FUNCTION_BLOCK AddRecipeToDatabase //IMPLEMENTS I_TcEventBase
VAR
	cmd : ARRAY[0..19] OF STRING_5K;
	query : STRING_5K;
	
	fbSQLCommand : FB_SQLCommandEvt(sNetID := '', tTimeout := T#5S);
	fbSQLDatabase : FB_SQLDatabaseEvt (sNetID := '', tTimeout := T#5S);
	fbSQLResult: FB_SQLResultEvt(sNetID:='', tTimeout:=T#5S);
	
	eventString : STRING_5K;
	
	step : (CONNECT, READY, EXECUTE, FINISH);
END_VAR
VAR_OUTPUT
	finished : BOOL;
END_VAR

CASE step OF
	CONNECT:
		IF fbSQLDatabase.Connect(1) THEN
			IF NOT fbSqlDatabase.bError THEN
				step := READY;
			END_IF
		END_IF
		
	READY:
		IF fbSQLDatabase.CreateCmd(ADR(fbSQLCommand)) THEN
			step := EXECUTE;
		END_IF
	
	EXECUTE:
		query := completeQuery();
		IF fbSQLCommand.Execute(ADR(query), SIZEOF(query)) THEN
			step := FINISH;
		END_IF
		
	FINISH:
		IF fbSQLDatabase.Disconnect() THEN
			finished := TRUE;
		END_IF
END_CASE

METHOD completeQuery : STRING_5K
VAR_INST
	reqProcess : ARRAY[0..3] OF STRING_5K;
	
	queryOpening : STRING_5K := 'INSERT INTO "Bundle Data - Prototype" (BundleID, Weight, Length, Height, Width, Pieces, Layers, PiecesPerLayer, ExtrusionWeight, ExtrusionHeight, ExtrusionWidth, RequiredProcesses, Paper_top, Paper_sides, Paper_bottom, Cardboard, CornerGuard, Chipboard, WoodBunk) VALUES (';;
	queryClosing : STRING_5K := ')';
END_VAR
reqProcess[0] := TO_STRING(BundleData.requiredProcessing[0]);
reqProcess[1] := TO_STRING(BundleData.requiredProcessing[1]);
reqProcess[2] := TO_STRING(BundleData.requiredProcessing[2]);
reqProcess[3] := TO_STRING(BundleData.requiredProcessing[3]);


cmd[0] := TO_STRING(BundleData.id);
CONCAT2(ADR('$''), ADR(cmd[0]), ADR(cmd[0]), SIZEOF(cmd[0]));
CONCAT2(ADR(cmd[0]), ADR('$''), ADR(cmd[0]), SIZEOF(cmd[0]));

cmd[1] := TO_STRING(BundleData.weight);
cmd[2] := TO_STRING(BundleData.length);
cmd[3] := TO_STRING(BundleData.height);
cmd[4] := TO_STRING(BundleData.width);
cmd[5] := TO_STRING(BundleData.pieces);
cmd[6] := TO_STRING(BundleData.layers);
cmd[7] := TO_STRING(BundleData.piecesPerLayer);

cmd[8] := TO_STRING(ExtrusionData.extrusionWeight);
cmd[9] := TO_STRING(ExtrusionData.extrusionHeight);
cmd[10] := TO_STRING(ExtrusionData.extrusionWidth);

cmd[11] := ConcatStrings(reqProcess, 'ARRAY[', ']', ',');
//strap wrap recipe
cmd[12] := paperQuery(StrapWrapRecipe.TopPaper); //Paper_top
cmd[13] := paperQuery(StrapWrapRecipe.LeftPaper); //Paper_sides
cmd[14] := paperQuery(StrapWrapRecipe.RightPaper); //Paper_sides
cmd[15] := paperQuery(StrapWrapRecipe.BottomPaper); //Paper_sides

cmd[16] := materialQuery(StrapWrapRecipe.Cardboard);
cmd[17] := materialQuery(StrapWrapRecipe.CornerGuard);
cmd[18] := materialQuery(StrapWrapRecipe.Chipboard);
cmd[19] := materialQuery(StrapWrapRecipe.WoodBunk);

completeQuery := ConcatStrings(cmd, queryOpening, queryClosing, ',');
END_METHOD

METHOD materialQuery : STRING_5K
VAR_IN_OUT
	materialArr : ARRAY[*] OF PositionMaterials;
END_VAR
VAR_INST
	tempQuery : STRING_5K;
	
	position : STRING;
	top : STRING;
	left : STRING;
	right : STRING;
	bottom : STRING;
	
	topLeft : STRING;
	topLeftFold : STRING;
	topRight : STRING;
	topRightFold : STRING;
	
	bottomLeft : STRING;
	bottomLeftFold : STRING;
	bottomRight : STRING;
	bottomRightFold : STRING;
	
	i : DINT;
END_VAR
tempQuery := 'ARRAY[';

FOR i:=LOWER_BOUND(materialArr, 1) TO UPPER_BOUND(materialArr, 1) BY 1 DO
	position := TO_STRING(materialArr[i].position);
	
	top := TO_STRING(materialArr[i].top);
	left := TO_STRING(materialArr[i].left);
	right := TO_STRING(materialArr[i].right);
	bottom := TO_STRING(materialArr[i].bottom);
	
	topLeft := TO_STRING(materialArr[i].topLeft);
	topRight := TO_STRING(materialArr[i].topRight);
	bottomLeft := TO_STRING(materialArr[i].bottomLeft);
	bottomRight := TO_STRING(materialArr[i].bottomRight);
	
	topLeftFold := TO_STRING(materialArr[i].topLeftFold);
	topRightFold := TO_STRING(materialArr[i].topRightFold);
	bottomLeftFold := TO_STRING(materialArr[i].bottomLeftFold);
	bottomRightFold := TO_STRING(materialArr[i].bottomRightFold);
	
	IF top = '' AND left = '' AND right = '' AND bottom = '' AND topLeft = '' AND topRight = '' AND bottomLeft = '' AND bottomRight = '' THEN
		CONTINUE;
	END_IF
	
	IF i > LOWER_BOUND(materialArr, 1) THEN
		CONCAT2(ADR(tempQuery), ADR(', '), ADR(tempQuery), SIZEOF(tempQuery));
	END_IF

	CONCAT2(ADR(tempQuery), ADR('('), ADR(tempQuery), SIZEOF(tempQuery));
	CONCAT2(ADR(tempQuery), ADR(position), ADR(tempQuery), SIZEOF(tempQuery));
	CONCAT2(ADR(tempQuery), ADR(',$''), ADR(tempQuery), SIZEOF(tempQuery));
	
	CONCAT2(ADR(tempQuery), ADR(top), ADR(tempQuery), SIZEOF(tempQuery));
	CONCAT2(ADR(tempQuery), ADR('$', $''), ADR(tempQuery), SIZEOF(tempQuery));
	CONCAT2(ADR(tempQuery), ADR(left), ADR(tempQuery), SIZEOF(tempQuery));
	CONCAT2(ADR(tempQuery), ADR('$', $''), ADR(tempQuery), SIZEOF(tempQuery));
	CONCAT2(ADR(tempQuery), ADR(right), ADR(tempQuery), SIZEOF(tempQuery));
	CONCAT2(ADR(tempQuery), ADR('$', $''), ADR(tempQuery), SIZEOF(tempQuery));
	CONCAT2(ADR(tempQuery), ADR(bottom), ADR(tempQuery), SIZEOF(tempQuery));
	CONCAT2(ADR(tempQuery), ADR('$', $''), ADR(tempQuery), SIZEOF(tempQuery));
	
	CONCAT2(ADR(tempQuery), ADR(topLeft), ADR(tempQuery), SIZEOF(tempQuery));
	CONCAT2(ADR(tempQuery), ADR('$', $''), ADR(tempQuery), SIZEOF(tempQuery));
	CONCAT2(ADR(tempQuery), ADR(topRight), ADR(tempQuery), SIZEOF(tempQuery));
	CONCAT2(ADR(tempQuery), ADR('$', $''), ADR(tempQuery), SIZEOF(tempQuery));
	CONCAT2(ADR(tempQuery), ADR(bottomLeft), ADR(tempQuery), SIZEOF(tempQuery));
	CONCAT2(ADR(tempQuery), ADR('$', $''), ADR(tempQuery), SIZEOF(tempQuery));
	CONCAT2(ADR(tempQuery), ADR(bottomRight), ADR(tempQuery), SIZEOF(tempQuery));
	CONCAT2(ADR(tempQuery), ADR('$', '), ADR(tempQuery), SIZEOF(tempQuery));
	
	CONCAT2(ADR(tempQuery), ADR(topLeftFold), ADR(tempQuery), SIZEOF(tempQuery));
	CONCAT2(ADR(tempQuery), ADR(', '), ADR(tempQuery), SIZEOF(tempQuery));
	CONCAT2(ADR(tempQuery), ADR(topRightFold), ADR(tempQuery), SIZEOF(tempQuery));
	CONCAT2(ADR(tempQuery), ADR(', '), ADR(tempQuery), SIZEOF(tempQuery));
	CONCAT2(ADR(tempQuery), ADR(bottomLeftFold), ADR(tempQuery), SIZEOF(tempQuery));
	CONCAT2(ADR(tempQuery), ADR(', '), ADR(tempQuery), SIZEOF(tempQuery));
	CONCAT2(ADR(tempQuery), ADR(bottomRightFold), ADR(tempQuery), SIZEOF(tempQuery));
	
	CONCAT2(ADR(tempQuery), ADR(')'), ADR(tempQuery), SIZEOF(tempQuery));
END_FOR
CONCAT2(ADR(tempQuery), ADR(']::"PositionMaterials"[]'), ADR(tempQuery), SIZEOF(tempQuery));

materialQuery := tempQuery;
END_METHOD

METHOD paperQuery : STRING_5K
VAR_IN_OUT
	paperArr : ARRAY[*] OF PaperInterval;
END_VAR
VAR_INST
	tempQuery : STRING_5K;
	i : DINT;
	start : STRING;
	end : STRING;
	wrap : STRING;
END_VAR
tempQuery := 'ARRAY[';

FOR i:=LOWER_BOUND(paperArr, 1) TO UPPER_BOUND(paperArr, 1) BY 1 DO
	start := TO_STRING(paperArr[i].start);
	end := TO_STRING(paperArr[i].end);
	wrap := TO_STRING(paperArr[i].wrap);
	
	IF start = '0' AND end = '0' AND wrap = 'FALSE' THEN
		CONTINUE;
	END_IF
	
	IF i > LOWER_BOUND(paperArr, 1) THEN
		CONCAT2(ADR(tempQuery), ADR(','), ADR(tempQuery), SIZEOF(tempQuery));
	END_IF

	CONCAT2(ADR(tempQuery), ADR('('), ADR(tempQuery), SIZEOF(tempQuery));
	CONCAT2(ADR(tempQuery), ADR(start), ADR(tempQuery), SIZEOF(tempQuery));
	CONCAT2(ADR(tempQuery), ADR(','), ADR(tempQuery), SIZEOF(tempQuery));
	CONCAT2(ADR(tempQuery), ADR(end), ADR(tempQuery), SIZEOF(tempQuery));
	CONCAT2(ADR(tempQuery), ADR(','), ADR(tempQuery), SIZEOF(tempQuery));
	CONCAT2(ADR(tempQuery), ADR(wrap), ADR(tempQuery), SIZEOF(tempQuery));
	CONCAT2(ADR(tempQuery), ADR(')'), ADR(tempQuery), SIZEOF(tempQuery));
END_FOR
CONCAT2(ADR(tempQuery), ADR(']::"PaperInterval"[]'), ADR(tempQuery), SIZEOF(tempQuery));

paperQuery := tempQuery;
END_METHOD

END_FUNCTION_BLOCK

(* stored: Version 1.1.0.1, ProductVersion 3.1.4024.11
   POU AddRecipeToDatabase: Id {63d7fce7-71e7-49a9-aa8c-4527f35d1303}, SpecialFunc None
   Folder Helpers: Id {d1d1d6bc-f89d-4d2d-843c-db59e83cb3f3}
   Method completeQuery: Id {05a935c7-eecf-4846-adb0-af86af87e8a3}
   Method materialQuery: Id {36340abb-1d4b-4d53-bb5a-85a0551c3552}
   Method paperQuery: Id {7cd757d5-fcc3-4d0d-bf77-ce348cc8c8e8} *)
